Staubli VAL3: initCmdBuf.pgx

program initCmdBuf()
  local num i
begin
  for i=0 to 19
    CmdBuffer[i]=""
  endFor
  CmdTotal=0
  nReadPt=0
  nWritePt=0
  //  setFrame(frm_ori,frm_x,frm_y,FrmDraw)
  jConfig=jHome
  libSave()
end
